FUNCTION F_LogDebug : STRING;
VAR_INPUT
	Message : T_MaxString;
END_VAR

F_LogDebug := 
	F_Logger( 
		E_LogSeverity.Debug, 
		CONCAT( 'DEBUG ' , Message ) 
	);

END_FUNCTION

(* stored: Version 1.1.0.1, ProductVersion 3.1.4022.18
   POU F_LogDebug: Id {adfe7a24-b378-4ac2-8722-b990d3e39262}, SpecialFunc None *)
